// TIA Portal V21 export
FUNCTION "GestStazione_ProntoInviare" : Void   // FC414, LAD
{ S7_Optimized_Access := 'TRUE' }
// stored: SetENOAutomatically false
   VAR_INPUT
      ProntoAdInviare : Bool;
      K_Stazione : Int;
   END_VAR
   VAR_TEMP
      DestinazioneAttuale : Int;
   END_VAR
BEGIN

REGION Network 1 (SCL): Codice necessario ad arrestare la chimata della destinazione a valle
   FOR #DestinazioneAttuale := 0 TO "K_NumStazione" DO //Sfoglio tutte le stazioni
       IF "Percorso".Stazione[#K_Stazione].Destinazione[#DestinazioneAttuale].IN.Attivo THEN   //Se la strada verso la destinazione è attiva (quindi selezionata e caricata in lavoro)
           IF NOT #ProntoAdInviare THEN                                                             //E ho il parametro in ingresso che chiede di fermare la destinazione
               "Percorso".Stazione[#DestinazioneAttuale].IN.SorgenteNonPronta := True;             //Fermo la destinazione
           END_IF;
       END_IF;
   END_FOR;
END_REGION
END_FUNCTION
